# EPICS autosave request: iocBoot/gmca_23i_ioc1/dbSave/MObm_Tn1_.req
%
% BURT Request File
%
% $(P)MO:Tn1:  Monochromator Crystal-1 tuning
%

file assy.req ASSY=$(P)MO:Tn1
file mtr1.req MTR1=$(P)MO:mr1
file drv1.req DRV1=$(P)MO:R1
